# B&R Automation Studio project TD52 (part 128)

### Module_MO.typ - Module global data types
```iecst
TYPE
	IN_MO_Struct : 	STRUCT
		tPB2MM : ParaBase2MM_type; (*Data exchange structure to ParaBase*) (*OldName:new PV; Cycle:5;*)
		iCANIdent : UDINT; (*CAN identifier from HalIO*) (*OldName:new PV; Cycle:2;*)
		bMisfCOn : BOOL; (*Misfire Command On *) (*OldName: MissfCmd; Cycle:5; *)
		tAB2MO : AmmBase2MM; (*AMM base to Monic data transfer*) (*OldName:QUITT_WA; Cycle:2;*)
	END_STRUCT;
	OUT_MO_Struct : 	STRUCT
		tMO2PB : MM2ParaBase_type; (*Data exchange structure to ParaBase*) (*OldName:new PV; Cycle:5;*)
		tMO2AB : MM2AmmBase; (*Monic module to AMM base data transfer*) (*OldName:new PV; Cycle:5;*)
		rU_IgnMon_Max : REAL; (*maximum ignition voltage *) (*OldName:MaxVolt; Cycle:5;*)
		rU_IgnMon_Min : REAL; (*minimum ignition voltage *) (*OldName:MinVolt; Cycle:5;*)
		iNum_IgnMon_Ver : INT; (*monic software version *) (*OldName:MonStatus; Cycle:5;*)
		rU_IgnMon_Cyl : ARRAY[0..24]OF REAL; (*ignition voltage for each cylinder *) (*OldName:V_Zyl; Cycle:5;*)
		tMonic_CanGo : CanDeviceGo; (*Start / Stop CAN communication*) (*OldName:new PV; Cycle:5;*)
		iMonicCommErrCount : USINT; (* counter comunication error monic *)
		iEMonStatus : USINT; (* event monic status *)
	END_STRUCT;
	_tMonicLimitREAL : 	STRUCT
		limit : REAL;
		kind : REAL;
		delay : REAL;
	END_STRUCT;
	_tMonicLimit : 	STRUCT
		limit : INT;
		kind : INT;
		delay : INT;
	END_STRUCT;
	CanDeviceGo : 	STRUCT
		CANDevGo : ARRAY[0..1]OF USINT; (*Start CAN communication and ID*)
		ECANDevGo : USINT; (*Wvent PV for start/stop communication*)
	END_STRUCT;
	MM2VIS_Struct : 	STRUCT
		rNum_IgnMon_Ver : REAL; (*Version of the firmware *) (*OldName:MonicVers; Cycle:;*)
		bMsg3201 : BOOL; (*W3201 MONIC CAN communication failure *) (*OldName:MONCAN; Cycle:;*)
		bMsg3202 : BOOL; (*W3202 MONIC CPU failure *) (*OldName:MONCPU; Cycle:;*)
		bMsg3203 : BOOL; (*W3203 MONIC wiring failure *) (*OldName:MONDRA; Cycle:;*)
		bMsg3181 : BOOL; (*W3203 MONIC AIC offset failure cylinder 1 *) (*OldName:MONOFF; Cycle:;*)
		bMsg3182 : BOOL; (*W3203 MONIC AIC offset failure cylinder 2 *) (*OldName:MONOFF; Cycle:;*)
		bMsg3183 : BOOL; (*W3203 MONIC AIC offset failure cylinder 3 *) (*OldName:MONOFF; Cycle:;*)
		bMsg3184 : BOOL; (*W3203 MONIC AIC offset failure cylinder 4 *) (*OldName:MONOFF; Cycle:;*)
		bMsg3185 : BOOL; (*W3203 MONIC AIC offset failure cylinder 5 *) (*OldName:MONOFF; Cycle:;*)
		bMsg3186 : BOOL; (*W3203 MONIC AIC offset failure cylinder 6 *) (*OldName:MONOFF; Cycle:;*)
		bMsg3187 : BOOL; (*W3203 MONIC AIC offset failure cylinder 7 *) (*OldName:MONOFF; Cycle:;*)
		bMsg3188 : BOOL; (*W3203 MONIC AIC offset failure cylinder 8 *) (*OldName:MONOFF; Cycle:;*)
		bMsg3189 : BOOL; (*W3203 MONIC AIC offset failure cylinder 9 *) (*OldName:MONOFF; Cycle:;*)
		bMsg3190 : BOOL; (*W3203 MONIC AIC offset failure cylinder 10 *) (*OldName:MONOFF; Cycle:;*)
		bMsg3191 : BOOL; (*W3203 MONIC AIC offset failure cylinder 11 *) (*OldName:MONOFF; Cycle:;*)
		bMsg3192 : BOOL; (*W3203 MONIC AIC offset failure cylinder 12 *) (*OldName:MONOFF; Cycle:;*)
		bMsg3193 : BOOL; (*W3203 MONIC AIC offset failure cylinder 13 *) (*OldName:MONOFF; Cycle:;*)
		bMsg3194 : BOOL; (*W3203 MONIC AIC offset failure cylinder 14 *) (*OldName:MONOFF; Cycle:;*)
		bMsg3195 : BOOL; (*W3203 MONIC AIC offset failure cylinder 15 *) (*OldName:MONOFF; Cycle:;*)
		bMsg3196 : BOOL; (*W3203 MONIC AIC offset failure cylinder 16 *) (*OldName:MONOFF; Cycle:;*)
		bMsg3197 : BOOL; (*W3203 MONIC AIC offset failure cylinder 17 *) (*OldName:MONOFF; Cycle:;*)
		bMsg3198 : BOOL; (*W3203 MONIC AIC offset failure cylinder 18 *) (*OldName:MONOFF; Cycle:;*)
		bMsg3199 : BOOL; (*W3203 MONIC AIC offset failure cylinder 19 *) (*OldName:MONOFF; Cycle:;*)
		bMsg3200 : BOOL; (*W3203 MONIC AIC offset failure cylinder 20 *) (*OldName:MONOFF; Cycle:;*)
		bMsg3204 : BOOL; (*W3204 MONIC parametering is running *) (*OldName:MONPAR; Cycle:;*)
		bMsg3208 : BOOL; (*W3208 MONIC firing voltage difference too high *) (*OldName:MONZ_D; Cycle:;*)
		bMsg3206 : BOOL; (*W3206 MONIC firing voltage too high *) (*OldName:MONZ_H; Cycle:;*)
		bMsg3207 : BOOL; (*W3207 MONIC average firing voltage too high *) (*OldName:MONZ_M; Cycle:;*)
		bMsg3205 : BOOL; (*W3205 MONIC firing voltage too low *) (*OldName:MONZ_N; Cycle:;*)
		iCMSinit_Monic_status : INT; (* Monic Module CMS Init Status *)
		iCMSmain_Monic_status : INT; (* Monic Module Main CMS Status *)
	END_STRUCT;
END_TYPE
```

### Module_MO.var - Module global variables
```iecst
VAR
	AvgVolt : UINT; (* ignition voltage average *)
	bGnlTrip_MO : BOOL := FALSE;
	bGnlTrip1_MO : BOOL := FALSE;
	bGnlTrip2_MO : BOOL := FALSE;
	bGnlTrip3_MO : BOOL := FALSE;
	bGnlWarning_MO : BOOL := FALSE;
	bInitOK : BOOL;
	CMSmain_Monic : CMSmain;
	CMSMonic_Init : CMSinit;
	DiffVolt : UINT; (* difference voltage monitoring Para_modlMO *)
	EConfMonic : ARRAY[0..67] OF USINT; (* event monic configuration *)
	ELimitErr : USINT; (* event monic limit errors *)
	EMonError : USINT; (* event monic device errors *)
	EMonStatus : USINT; (* event monic status *)
	EnabGuard : USINT; (* parameter enable guarding *)
	EnabLimit : USINT; (* parameter enabel limit monitoring *)
	EnabMonic : USINT; (* operating mode monic *)
	FGDRPS : BOOL; (* Freigabe durch RPS *)
	iECanDevGo : DINT;
	Ignor : ARRAY[0..24] OF BOOL; (* TRUE= ignor cyl. limit monitoring *)
	IN_MO : IN_MO_Struct;
	LimitActiv : USINT; (* ignition voltage start monitoring *)
	LimitError : UINT; (* status of voltage limit errors *)
	LimitHyst : USINT; (* hysteresis for start monitoring *)
	LimitMon : ARRAY[0..4] OF _tMonicLimit; (* parameter voltage limit monitoring *)
	MaxVolt : UINT; (* maximum ignition voltage *)
	MinVolt : UINT; (* minimum ignition voltage *)
	MissfCmd : BOOL; (* command for start misfire *)
	MM2VIS : MM2VIS_Struct := (0);
	Mon_Node : USINT; (* node number monic *)
	MONCAN : BOOL := 0; (* CAN VUS FAHLER *)
	MONCPU : BOOL := 0; (* MONIC CPU FEHLER *)
	MONDRA : BOOL := 0; (* MONIC VERDRAHTUNGSFEHLER *)
	monic_vis : BOOL; (* TRUE= monic is enabled *)
	MonicError : ARRAY[0..6] OF USINT; (* monic error messages *)
	MonLimitOn : ARRAY[0..4] OF BOOL; (* type of voltage limit monitoring *)
	MONOFF : ARRAY[0..24] OF BOOL := [25(0)]; (* MONIC AIC ODDSET FEHLER *)
	MONPAR : BOOL := 0; (* MONIC PAREMETRIERUNG IM BETRIEB *)
	MonStatus : ARRAY[0..4] OF USINT; (* monic status message *)
	MONZ_D : BOOL := 0; (* MONIC ignition voltage difference*)
	MONZ_H : BOOL := 0; (* MONIC ignition voltage too high*)
	MONZ_M : BOOL := 0; (* MONIC ignition voltage average*)
	MONZ_N : BOOL := 0; (* MONIC ignition voltage too low*)
	OUT_MO : OUT_MO_Struct;
	Para : PARA_MO_Struct;
	ParaFactoryDefault : PARA_MO_Struct := (0);
	pm : PARA_MO_Struct;
	TrigVolt : USINT; (* tirgger voltage for volt. measure *)
	ucEAvgVolt : USINT; (* event average cylinder voltage *)
	ucEDifVolt : USINT; (* event cylinder voltage difference *)
	ucEMaxVolt : USINT; (* event maximum cylinder voltage *)
	ucEMinVolt : USINT; (* event minimum cylinder voltage *)
	ucEV_Zyl : ARRAY[0..24] OF USINT; (* event actual cylinder voltage *)
	ucMonicCommErrCount : USINT; (* counter comunication error monic *)
	usV_Zyl : ARRAY[0..24] OF UINT; (* ignition voltage for each cylinder *)
	xEngtype : EngType; (*FB for Engine type specific values*)
	ZylZahl : USINT;
	FireOrder : ARRAY[0..24] OF USINT;
	bNoInitDetected : BOOL := FALSE; (*allways true, except 1cycle on init up*)
	ucCountG : USINT;
END_VAR
```

### Module_MOPara.typ - Module global parameter
```iecst
TYPE
	PROGRAMMER_INFO : 	STRUCT
		DO_NOT_SORT_PARA : STRING[40] := 'DO NOT CHANGE PARAMETER SORTING!'; (*DO NOT CHANGE PARAMETER SORTING!*) (*ADD NEW PARAMETER ONLY AT THE END OF THE Para STRUCTURE. DO NOT DELETE existing Para items.*)
	END_STRUCT;
	PARA_MO_Struct : 	STRUCT
		iEng_Motortype : INT; (*PARA: engine motortype*) (*OldName:Motortype; Cycle:;*)
		rU_IgnMon_LimActive : REAL; (*PARA [12155]: ignition voltage start monitoring *) (*OldName:LimitActiv; Cycle:;*)
		rU_IgnMon_LimHy : REAL; (*PARA [12088]: hysteresis for start monitoring *) (*OldName:LimitHyst; Cycle:;*)
		bIgnMon_Active : BOOL; (*PARA [12064]: TRUE= monic is enabled *) (*OldName:monic_vis; Cycle:;*)
		iU_Ign_LimMonTrig : INT; (*PARA [12087]: trigger voltage for volt. measure *) (*OldName:TrigVolt; Cycle:;*)
		bIgn_LimitMonitorActive : ARRAY[0..4]OF BOOL; (*Para: Type of voltage limit monitoring*) (*OldName:MonLimitOn; Cycle:;*)
		tIgn_LimitMonitor : ARRAY[0..4]OF _tMonicLimitREAL; (*Para: Ignition voltage monitoring*) (*OldName:LimitMon; Cycle:;*)
		zz_V4_0_ParaVersionEnd : REAL := 4.01; (*! ADD NEW PARAMETER ONLY BELOW THIS LINE ! This is the end of base version parameter and has to stay unchanged. DO NOT CHANGE SORT ORDER of Para!*) (* OldName: new PV; Cycle: 5; *)
	END_STRUCT;
END_TYPE
```

- Logical/Monic/monic (protected, skipped)

### Program Logical/Monic/IN_MO (IEC, version 4.00.2) - + IN task

- IN_MOCyclic.st (not readable text: treated as protected, skipped)

### Program Logical/Monic/OUT_MO (IEC, version 4.05.0) - + OUT task

- OUT_MOCyclic.st (not readable text: treated as protected, skipped)

### Program Logical/Monic/MsgMO (IEC, version 4.00.0) - + Messages

- MsgMOCyclic.st (not readable text: treated as protected, skipped)

- MsgMOInit.st (not readable text: treated as protected, skipped)

#### MsgMO.var - Local variables
```iecst
VAR
	iAdrAmmBase2MM : UDINT;
	iAdrMM2AmmBase : UDINT;
	xMsg3201 : Msg;
	xMsg3202 : Msg;
	xMsg3203 : Msg;
	xMsg3204 : Msg;
	xMsg3205 : Msg;
	xMsg3206 : Msg;
	xMsg3207 : Msg;
	xMsg3208 : Msg;
	xMsg3181 : Msg;
	xMsg3182 : Msg;
	xMsg3183 : Msg;
	xMsg3184 : Msg;
	xMsg3185 : Msg;
	xMsg3186 : Msg;
	xMsg3187 : Msg;
	xMsg3188 : Msg;
	xMsg3189 : Msg;
	xMsg3190 : Msg;
	xMsg3191 : Msg;
	xMsg3192 : Msg;
	xMsg3193 : Msg;
	xMsg3194 : Msg;
	xMsg3195 : Msg;
	xMsg3196 : Msg;
	xMsg3197 : Msg;
	xMsg3198 : Msg;
	xMsg3199 : Msg;
	xMsg3200 : Msg;
END_VAR
```

### Program Logical/Monic/ParMO (IEC, version 4.06.0) - + Parameter handling

- perm_par.st (not readable text: treated as protected, skipped)

#### perm_par.var
```iecst
VAR
	tParaIntern : ParaHandler_typ; (*Connector type to perm_par*)
	tMM2ParaBase_ReadBack : MM2ParaBase_type; (*INTERNAL! V4.06 new readback structure for information from previous tasks*)
	bWriteDataObj : BOOL; (* TRUE=write data object module *)
	bDataObjLenErr : BOOL; (*Error occured in permem: data module size missmatch*)
	bCreateDataObj : BOOL; (* TRUE=create new data object *)
	bWriteOnce : BOOL; (* write permanent memory once *)
	DatObjCreate_01 : DatObjCreate; (* data object create *)
	DatObjInfoBak_02 : DatObjInfo; (* data object info *)
	DatObjDelete_01 : DatObjDelete; (* data object delete *)
	DatObjRead_01 : DatObjRead; (* data object read *)
	DatObjRead_02 : DatObjRead; (* manual initiated data object read *)
	DatObjWrite_01 : DatObjWrite; (* data object write *)
	DatObjDelete_02 : DatObjDelete; (* data object delete *)
	DatObjDelete_11 : DatObjDelete; (*Delete Backup File*)
	DatObjInfo_01 : DatObjInfo; (* data object info *)
	DatObjInfo_02 : DatObjInfo; (* data object info *)
	szModuleName : STRING[35]; (* module name of object *)
	szModuleNameBackup : STRING[35]; (* module name of posiibly created backup object *)
	DatObjCopy_01 : DatObjCopy;
	bCopyDataObj : BOOL;
	TON_WarnDelay : TON;
	TON_WritePMEM : TON; (* delay write permanent memory *)
	ulPMPointer : UDINT; (* adress of actual checksum value *)
	ulChecksum : UDINT; (* parameter checksum value *)
	pm_len : UDINT; (* permanent value lenght *)
	ulChecksumOld : UDINT; (* last vlaue of parameter checksum *)
	ulChkValue : UDINT; (* actual value of parameter pointer *)
	pm_id : UDINT; (* permanent value identifier *)
	pm_p : UDINT; (* permanent value pointer *)
	DatObjInfo_META : DatObjInfo;
	DatObjRead_META : DatObjRead;
	szMetaDataRaw : STRING[2000];
	szMetaData : ARRAY[0..4] OF STRING[35];
	szMetaDataVis : ARRAY[0..3] OF STRING[35];
	ssIndex : INT;
	ssCount : INT;
	ucMetaDataRaw : ARRAY[0..2000] OF USINT;
	ssCount2 : INT;
	szMetaDataFile : STRING[10];
	szText1 : STRING[20];
	pv_adr_IN_XX_tPB2MM : UDINT;
	pv_lng : UDINT;
	pv_lng_IN_XX_tPB2MM : UDINT;
	pv_lng_OUT_XX_tPB2MM : UDINT;
	szText2 : STRING[20];
	pv_adr_OUT_XX_tXX2PB : UDINT;
END_VAR
VAR CONSTANT
	ERR_NOERROR : UINT := 0;
END_VAR
VAR
	usPMWriteCnt : UINT;
	pm_Error : UDINT; (* permanent value error *) (* Deleted: pm : ParaMem_typ; permanent memory tags mathias, 22.8.11*)
	fun_Error : UDINT := 0; (*state > 0 = function error*)
	xLocalParaCheck : ParaCheckFUB; (*local function instance to check parameter values*)
	TON_ParaSetupOk : TON;
	bParaCheckSystemOk : BOOL;
	iDebug_ParaOkChecked : UDINT;
	bRestoreBackupDataObj : BOOL := FALSE;
	bRestoreDataObjContent : BOOL := FALSE;
	pm_id_backup : UDINT;
	pm_p_Backup : UDINT;
	DatObjCopy_02 : DatObjCopy;
	bDeleteBackupDataObj : BOOL := FALSE; (*Command to delete backup data module file on purpose*)
	bDebugPara : ARRAY[0..5] OF BOOL;
	ssIndex2 : INT;
	ssIndex3 : INT;
	ssIndex4 : INT;
	ssIndexVis : INT;
	szText : STRING[40];
	pv_adr_Para : UDINT;
	szParaSnippet : ARRAY[0..5] OF STRING[150];
	szParaIndex : STRING[10];
	slValue : DINT;
	iModuleDLD_ResetCount : INT;
	bDownloadDetected : BOOL;
	bFlagParaStructCopyWorking : BOOL; (*true, if cyclic para copying is active, 1 false cycle at every copy *)
	bStoreInitParaInDataObj : BOOL := FALSE;
	bTestflag : BOOL;
	bReadOutMETA_Once : BOOL;
	tParaCheck_iPvAdress : ARRAY[0..5] OF UDINT;
	tParaCheck_iPvLengt : ARRAY[0..5] OF UDINT;
	tParaCheck_rPvValue : ARRAY[0..5] OF REAL;
	tParaCheck_rRangeMIN : ARRAY[0..5] OF REAL;
	tParaCheck_rRangeMAX : ARRAY[0..5] OF REAL;
	tParaCheck_szPvName : ARRAY[0..5] OF STRING[35];
	ssFormatDetected : INT;
	szMetaDataPart : STRING[150];
	szFullTaskName : STRING[35];
	szFullMetaModuleName : STRING[35];
	debugLen : INT;
	debugSize : INT := 0;
	strcat_adr1 : UDINT;
	strcat_adr2 : UDINT;
	ssIndexTN : INT;
	bAlternate : BOOL;
	n : INT;
	iAlternateChecksum : DINT;
	iAlternateChecksumOld : DINT;
	ulDebugChkValue : ARRAY[0..999] OF UDINT;
	Adr1 : UDINT;
	Adr2 : UDINT;
	usPMWriteCntStepsize : UINT := 1; (*different step sizes to help debug*)
	usPMWriteCntXOR : UINT;
	usPMWriteCntAltSum : UINT;
	ulAdrPM : UDINT;
	usChkValuePM : USINT;
	ulAdrPara : UDINT;
	ulPara_len : UDINT;
	usChkValuePara : USINT;
	iDebugCountPMDifferences : DINT := 0;
	bEngineRunDetected : BOOL; (*detection status bit autocommand 100 /101  for engine run state*)
	ucMetaDataDebugInfoLine : ARRAY[0..24] OF STRING[80];
	ssIndexMand : INT := 0;
	szMetaDataMand : STRING[35];
	iMyErrorInfo_Autoreset : DINT; (*internal autoreset counter*)
	ssIndex_Version : INT; (*internal*)
	ssIndex_BU : INT; (*internal*)
	ssIndex_BU2 : INT; (*internal*)
END_VAR
```


### Package Logical/Opstate - OP: Operation State

### Data object Logical/Opstate/META_OP (Simple) - Simple data object.

#### META_OP.dat
```
; *******************************************************************************
; AGGR: Module Meta Data (data module)
;
; This code is confidential and proprietary to the INNIO Company.
; It may not be used in any form, or reproduced in any manner, without the express
; written permission of the INNIO Company.
; Copyright, INNIO Company, 2023
;
; Customized modifications: -
; ------------------------
;
; History:
; -------
; V3.99	06-03-2013	Weitzer, generated for modular software
; V4.00 31.01.2014	Weitzer, versions changed
; V4.00 10.02.2014	Graus, 	 change module function description and dependencies
; V4.01 22.07.2104	Weitzer, increase version number --> new reserve P limitation added
; V4.02 25.02.2015	Graus, 	 increase version number, add dependency from SAFI module
; V4.02.1  	11.06.2015	Zengerer	 version + dependencies changed (IF change with array index 0 for compatibility with c-tasks)
; V4.04.00 	12.07.2016	502423184	versions changed
; V4.05.01	25.09.2017 	Gomez Ortiz Removal of UW_PDIFF_A (engine type dependency) from the Alarm 1108 and 2097 Alarm
; V4.05.01	01.03.2018	Perktold	Korrektur bOpM_Pr_CC_Hi fuer globale Pred Anzeige
; V4.05.02	05.04.2018	Perktold	OPState: added IN_OP.bFS_Act for OilSkid Start Release Type 9
; V4.05.02	05.09.2018	Zuschnig,	BU 01: Correction ramp for demand off - gridcode
; V4.05.02	05.09.2018	Gwiggner	BU 01: bugfix function block xTP_OpenGV;
; V4.06.00	20.09.2018	Perktold	changes for GEN2/FastStart
; V4.07.00	26.04.2018	lettenb.	SWAT920/5 added
; V4.07.01	04.05.2018	502423184,	added fast power reduction to out interface
; V4.07.02	23.07.2018	Messner		CPP Integrator power reduction added
;			14.01.2019	Schmid		W9249 (deflagration detection) blocks engine restart
; V4.07.03	31.01.2019	502423184	new Opstate, Powersel and Speedsel
; V4.07.04	29.03.2019	Hohensinner	Bugfixing: TPSA Library, added missing interface to VIS for PRed CppInt, added W9284, added ramp for power set point in droop mode
; V4.07.05	15.05.2019	Hohensinner	added EngBlock_PlantCtr DI --> Blocks module smooth & W1188, converted new Parameter from rTi (REAL) to ti (TIME) (coding guideline)
; 			04.11.2019	Schmidt		BU 01: Type 6 cooldown run duration modified from 0s to 10s, div by 0
; V4.09.00	03.02.2020	Zuschnig	TOF in TPSA Library always active, included TOF (60s) for operation message B1283 to B1287
;			12.02.2020	Zuschnig	Included ParaSetupOk plus 2 sec to release power reductions and B2140, included B2972 and B2973 - Power Mode on/off
; V4.10.00	22.05.2020	lettenb.	bEng_Bloc[29-33] added
;			20.10.2020	Zuschnig	removed activation of module blocked by oil skid only if fast start is active -> always active
; 			21.10.2020	Zuschnig	Add speed adjustment for resynchronization with MMD2
; 			16.10.2020  Weitzer		release P reduction at Load Sharing Line by customer bus signal IN_OP.bRel_P_Red_I_Bus
;									release speed control by cusotmer bit IN_OP.bN_U_Set_Ext_On
;									release power mode by customer bit IN_OP.bReq_PowMod_Ext
;       	10.12.2020	Zuschnig	Included power reduction for Tecjet differential pressure
;			18.01.2021	Perktold	unbundling emergency stop and fire alarm
;	     	20.01.2021	Zuschnig	increased max. sy delta speed to -0.06 (from -0.05)
;			20.01.2021  Zuschnig	Included maximum for power ramp increase and decrease
;			24.03.2021  Gwiggner	delay of LSL by 300ms
; V4.11.00	21.05.2021  Zuschnig	Bugfix - B2154 triggered with high frequency bit
;           16.08.2021	Keller		Droop Mode Power Controller, Overload Protection in Isolated Operation
;			16.11.2021	Andre		Added SAFI config done bit to the startup release
;			22.11.2021	Perktold,	added myPlant remote request/P-setpoint
;			22.12.2021	Andre		Added Power reduction by CAN communication failure for half or more SAFI or too many SAFI reboots
;			15.03.2022	Zuschnig	Deactivate power ramp when GCB is opened
;			01.04.2022	Zuschnig 	TOF with 60s for messages 2130, 2152, 2153 and 2154 to prevent too many messages
; V4.12.00	01.08.2022	Zuschnig	Speed offset selection for AB Energy
;			19.08.2022	Keller		Limit LSL speed reference offset to +-3.3%Nnom
;			08.09.2022	Andre		Added SEMIC config done bit to the startup release
;			26.09.2022	Perktold	Added IN signal to xTOFIgn_Dem in case of a prio 1 trip
;			22.01.2023	Zuschnig	Increased max. sy delta speed for IN_OP.bSynchDem
;			22.01.2023  Zuschnig	Include power reduction H2 content
;			25.01.2023	Tinello		Deleted power reduction by T1HP / Added power reduction by T2HP and T2LP / Added engine blocked by charge temperature after TC
; V4.13.00  14.04.2023  Bachler     Add overload and reverse power protection in isolated operation
;       	05.07.2023	Zuschnig	Removed Step Time Display Information
;			26.09.2023	Farre,		Addition engine blocked by LCB opened (info #37)
;           16.10.2023  Bachler     Changed initialization of LSL when switching to LSL speed mode for bumpless transition
;           17.10.2023  Bachler 	Add integrator to compensate for signal errors of the load sharing line
;			03.11.2023	Zuschnig	Add operating counter low load
;			20.11.2023	Zengerer	Add counter correction IN_OP.iCnt_OpHours_Set, iCnt_UnitOpHours_Set, iCnt_FastStarts_Set, iCnt_FastStarts_Set
;			20.11.2023	Farre,		added "request power mode" interface; extended operating range (IN_OP.rP_Set_Min_Norm) (2023-168)
;       	03.07.2023	Goenczi		Adaptions for Aggreko serialization
;			17.01.2024	Schmidt		Bugfix deflagration protection: added IN_OP.bIgnDeflPrct_Off to ignition demand logic (issue 1406)
; 			26.01.2024 	Zuschnig 	Bugfix FPR during demand off
; V4.14.00	28.03.2024	Soto/Farre,	Added CAN WG configuration for start up release (2023-174)
;			25.10.2024	Farre		include in bEng_Bloc[1] - rel. sync - when GCB position signal failure and enigne stopped (2024-241)
;			25.11.2024	Bacci		T6 Start procedure with purge start (2024-219): added waiting time for starter release in state 32 and 7
;			28.11.2024	Kafka		remove power reduction from LHE
; 			29.11.2024	Farre		calculation of power reduction due to CosPhi <1, from OP to GC (issue #1700)
;
; Instructions for use:
; --------------------
; make only changes at the version numbers
;
; Outstandings:
; ------------
;
; *******************************************************************************
;
"<META>"
;
; Module ID
"<MODUL>OP</MODUL>"
;
; Module Version (xx.yy.zz.cc)
"<VERSION>04.14.00.00</VERSION>"
;
; Module Basisupdate Version BU (00-99)
"<BASISUPDATE_VERSION>00</BASISUPDATE_VERSION>"
;
; Optional: specify order number for limitated module usage
"<ORDER></ORDER>" ;<!--(optional for restricted customizations; missing statement makes module valid for all orders)-->
;
; Parameter Check <PARAn Name='aAbcdef' MIN='xxx' MAX='yyy' />  (watch for correct spacings and apostrophs!)
"<PARAMETER_CHK>"
"<PARA1 Name='iEng_Motortype' MIN='208' MAX='920' />"
"<PARA2 Name='rN_EngNom' MIN='100.0' MAX='2000.0' />"
"<PARA3 Name='rP_Nom_Gastype[1]' MIN='10.0' MAX='15000.0' />"
"<PARA4 />"
"<PARA5 />"
"</PARAMETER_CHK>"
;
; Statement, that this module´s parameter check passing is mandatory (OP is allways mandatory, so other statements than TRUE here in this module are ignored)
"<MANDATORYMODULE>TRUE</MANDATORYMODULE>"
;
; Permanent Datamodule Filenames<!-- NAME ist ohne Dateiendung einzutragen; Nur für Counter und interne Parameter verwenden-->
"<DATAMODULES>" ;<!-- optional; mehrere DATAMODULES erlaubt-->
"	<DATAMODULE>par_OP</DATAMODULE>"
"	<DATAMODULE>perm_OP</DATAMODULE>"
"</DATAMODULES>"
;
; Dependencies Modules (MMxx.yy.zz.cc)
"<DEPENDENCIES>"
"	<DEPENDENCY MODULE='HA' VERSION='04.10.00.00' />"
"	<DEPENDENCY MODULE='GT' VERSION='04.12.00.00' />"
"	<DEPENDENCY MODULE='AG' VERSION='04.14.00.00' />"
"	<DEPENDENCY MODULE='EC' VERSION='04.14.00.00' />"
"	<DEPENDENCY MODULE='IG' VERSION='04.00.00.00' />"
"	<DEPENDENCY MODULE='SY' VERSION='04.14.00.00' />"
"	<DEPENDENCY MODULE='EX' VERSION='04.10.00.00' />"
"	<DEPENDENCY MODULE='EG' VERSION='04.00.00.00' />"
"	<DEPENDENCY MODULE='HC' VERSION='04.00.00.00' />"
"	<DEPENDENCY MODULE='KN' VERSION='04.00.00.00' />"
"	<DEPENDENCY MODULE='CH' VERSION='04.05.00.00' />"
"	<DEPENDENCY MODULE='VE' VERSION='04.00.00.00' />"
"	<DEPENDENCY MODULE='GC' VERSION='04.14.00.00' />"
"	<DEPENDENCY MODULE='CU' VERSION='04.13.00.00' />"
"	<DEPENDENCY MODULE='GR' VERSION='04.00.00.00' />"
"	<DEPENDENCY MODULE='CP' VERSION='04.00.00.00' />"
"	<DEPENDENCY MODULE='PB' VERSION='04.13.00.00' />"
"	<DEPENDENCY MODULE='AB' VERSION='04.00.00.00' />"
"	<DEPENDENCY MODULE='GM' VERSION='04.01.00.00' />"
"	<DEPENDENCY MODULE='SA' VERSION='04.11.00.00' />"
"	<DEPENDENCY MODULE='IC' VERSION='04.12.00.00' />"
"   <DEPENDENCY VISVERSION='02.15.00.00' />"			; Dependencies Visualization
"</DEPENDENCIES>"
;
; Module function description
"<MODULEFUNCTION>" ;<!-- short overview documentation of module function; add reference to detailed information, if available-->
"	<General>	"
"	Handling of engines operation mode "
"	</General>	"
""
"	<F1 Name='Engine state machine' LastModified='4.0.2.0'>"
"	State machine to determine engines operation mode.	"
"	</F1>"
"	<F2 Name='Power set value' LastModified='4.0.2.0'>"
"	Determination the power set value concerning the load ramp gradients and the load reductions.	"
"	</F2>"
"	<F3 Name='Speed set value' LastModified='4.0.0.0'>"
"	Determination of the engine speed set value for idle- and isolated operation mode.	"
"	</F3>"
"	<F4 Name=' frequency control' LastModified='4.2.0.1'>"
"   changed priority order of power setpoint change 	"
"	</F4>"
""
"	<Info>"
" 	UPDATE V4.01.01.00  Perm datamodule moved from SYS- to USERROM	"
"   UPDATE V4.02.01.00	version + dependencies changed (IF change with array index 0 for compatibility with c-tasks)	"
" 	UPDATE V4.04.00.00  delayed version of State32 "
"	UPDATE V4.05.02.00  BU 01: Correction ramp for demand off - gridcode "
"	UPDATE V4.05.02.00	BU 01: bugfix function block xTP_OpenGV "
"	UPDATE V4.07.05.00	BU 01: Type 6 cooldown run duration modified from 0s to 10s, div by 0"
"	UPDATE V4.11.00.00	Bugfix - B2154 triggered with high frequency bit"
"	UPDATE V4.13.00.00	Add counter correction IN_OP.iCnt_OpHours_Set, iCnt_UnitOpHours_Set, iCnt_FastStarts_Set, iCnt_FastStarts_Set "
"	</Info>"
""
"	<Customized LastModified='4.0.0.0'>	"
"	- Nothing "
"	</Customized>	"
""
"</MODULEFUNCTION>"
;
"</META>"
```
